// TIA Portal V17 export
// export: Created 2025-06-25T13:13:07.6103619Z, ExportSetting WithDefaults, DisplayName Totally Integrated Automation Portal, DisplayVersion V17 Update 8, DisplayName TIA Portal Openness, DisplayVersion V17 Update 8, DisplayName TIA Portal Version Control Interface, DisplayVersion V17, DisplayName STEP 7 Professional, DisplayVersion V17 Update 8, DisplayName STEP 7 Safety, DisplayVersion V17 Update 6, DisplayName WinCC Advanced, DisplayVersion V17 Update 8
FUNCTION_BLOCK "SuperheatControl"   // FB23, FBD
TITLE = Pinch setpoint from superheat
{ S7_Optimized_Access := 'TRUE' }
VERSION : 0.1
// stored: AutoNumber true, IsIECCheckEnabled false, IsRetainMemResEnabled false, MemoryReserve 100, SetENOAutomatically false, UDAEnableTagReadback false
   VAR_INPUT
      bEnable { ExternalAccessible := 'False'; ExternalVisible := 'False'; ExternalWritable := 'False'} : Bool;   // 1 = enable controller 0 = disable controller
      bReset { ExternalAccessible := 'False'; ExternalVisible := 'False'; ExternalWritable := 'False'} : Bool;   // 1 = reset manual mode
      AdditionalSuperheat { ExternalAccessible := 'False'; ExternalVisible := 'False'; ExternalWritable := 'False'} : Real;
   END_VAR
   VAR_OUTPUT
      AddSuperheat { ExternalAccessible := 'False'; ExternalVisible := 'False'; ExternalWritable := 'False'} : Real;
   END_VAR
   VAR
      SuperheatSetpoint { ExternalAccessible := 'False'; ExternalVisible := 'False'; ExternalWritable := 'False'} : Real;
      PinchSetpoint { ExternalAccessible := 'False'; ExternalVisible := 'False'; ExternalWritable := 'False'} : Real;
      PinchPerformanceCurrent { ExternalAccessible := 'False'; ExternalVisible := 'False'; ExternalWritable := 'False'} : Real;
      Regulator { ExternalAccessible := 'False'; ExternalVisible := 'False'; ExternalWritable := 'False'} : Struct
         x_intern_1 { ExternalAccessible := 'False'; ExternalVisible := 'False'; ExternalWritable := 'False'} : Real;
         x_intern_2 { ExternalAccessible := 'False'; ExternalVisible := 'False'; ExternalWritable := 'False'} : Real;
         x_intern_3 { ExternalAccessible := 'False'; ExternalVisible := 'False'; ExternalWritable := 'False'} : Real;
      END_STRUCT;
      Enabled { ExternalAccessible := 'False'; ExternalVisible := 'False'; ExternalWritable := 'False'} : Bool;
      A3020 { ExternalAccessible := 'False'; ExternalVisible := 'False'; ExternalWritable := 'False'} : "fbHMIEvent";
   END_VAR
   VAR_TEMP
      PinchPerformance : Real;
      PIDControlInactive : Bool;   // Is true if pinch setpoint is externally controlled
   END_VAR
BEGIN

REGION Network 1: Reset manual mode
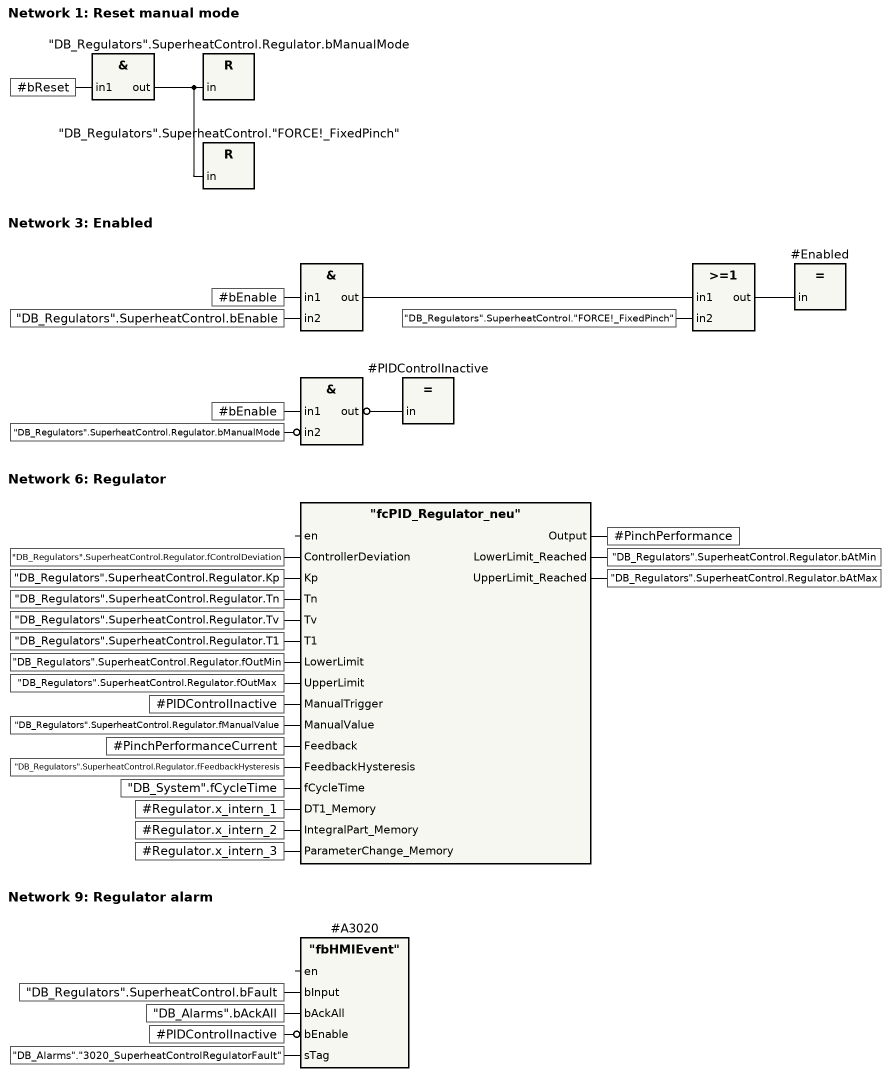
   IF #bReset THEN
       "DB_Regulators".SuperheatControl.Regulator.bManualMode := FALSE;
       "DB_Regulators".SuperheatControl."FORCE!_FixedPinch" := FALSE;
   END_IF;
END_REGION

REGION Network 2 (SCL): Manual values are given as Pinch, regulator works on "Pinch Performance"
   "DB_Regulators".SuperheatControl.Regulator.bManualMode := "DB_Regulators".SuperheatControl."FORCE!_FixedPinch";
END_REGION

REGION Network 3: Enabled
   // NOTE that we are not using the conventional bManual bit!!
   // Due to the difference between "Pinch Performance" and "Pinch"
   #Enabled := (#bEnable AND "DB_Regulators".SuperheatControl.bEnable) OR "DB_Regulators".SuperheatControl."FORCE!_FixedPinch";
   #PIDControlInactive := NOT (#bEnable AND NOT "DB_Regulators".SuperheatControl.Regulator.bManualMode);
END_REGION

REGION Network 4 (SCL): Superheat setpoint
   //Additional Superheat
   #AddSuperheat := #AdditionalSuperheat + "DB_Regulators".SuperheatControl.AdditionalSuperheat + "DB_CurrentSetting".Fluid.T_AdditionalSuperHeatEvaporator;

   #SuperheatSetpoint := 1.0 * "RecTarget"("DB_Regulators".SuperheatControl.fineTuningRecTarget) +
                         1.0 * #AddSuperheat;

   // Superheat setpoint
   IF "DB_State".State."6_Running" THEN
       #SuperheatSetpoint := #SuperheatSetpoint + 1.0 * "VapPerformance"(AddSuperheat := #AddSuperheat, Pinch := #PinchSetpoint);
   ELSE
       #SuperheatSetpoint := #SuperheatSetpoint + 0.5 * "VapPerformance"(AddSuperheat := #AddSuperheat, Pinch := #PinchSetpoint);

   END_IF;

   // Enforce a lower bound on the superheat
   #SuperheatSetpoint := MAX(IN1 := #SuperheatSetpoint, IN2 := "DB_CurrentSetting".System.Limits.T_SuperHeatCompressorIn_Min + 5.5);
END_REGION

REGION Network 5 (SCL): Deviation
   IF "DB_Regulators".SuperheatControl.Regulator.bManualMode = TRUE THEN
       "DB_Regulators".SuperheatControl.Regulator.fManualValue := LN(MAX(IN1 := "DB_Regulators".SuperheatControl."FORCE!_FixedPinch_Value", IN2 := 0.01)) * "DB_Regulators".SuperheatControl.ExponentialPinchFactor;
       "DB_Regulators".SuperheatControl.bFault := FALSE;
   ELSE
       //- Preset manual value to current pinch value to set controller to this value if inactive. Except if bManualMode whwre we directely set it to the target pinch performance
       //- Limited to 1K superhetat to prevent division by zero and critical low pinch values
       "DB_Regulators".SuperheatControl.Regulator.fManualValue := LN(MAX(IN1 := "DB_Calc".HeatSource.Pinch.fValue, IN2 := 1)) * "DB_Regulators".SuperheatControl.ExponentialPinchFactor;

       //Preset with current pinch as starting value if "FORCE!_FixedPinch is used
       "DB_Regulators".SuperheatControl."FORCE!_FixedPinch_Value" := "DB_Calc".HeatSource.Pinch.fValue;


       //Auto mode setpoint
       IF "isNaN"("DB_Calc".LowPressPart.CompressorSuperheat.fValue) OR "isNaN"(#SuperheatSetpoint) THEN
           "DB_Regulators".SuperheatControl.Regulator.fControlDeviation := 0;
           "DB_Regulators".SuperheatControl.bFault := TRUE;
       ELSE
           "DB_Regulators".SuperheatControl.Regulator.fControlDeviation := #SuperheatSetpoint - "DB_Calc".LowPressPart.CompressorSuperheat.fValue;
           "DB_Regulators".SuperheatControl.bFault := FALSE;
       END_IF;
   END_IF;

   //- Current pinch performance for informative reasons
   //- Limited to 0.1K to prevent division by zero 
   #PinchPerformanceCurrent := LN(MAX(IN1 := "DB_Calc".HeatSource.Pinch.fValue, IN2 := 0.1)) * "DB_Regulators".SuperheatControl.ExponentialPinchFactor;
END_REGION

REGION Network 6: Regulator
   "fcPID_Regulator_neu"(ControllerDeviation := "DB_Regulators".SuperheatControl.Regulator.fControlDeviation,
                         Kp := "DB_Regulators".SuperheatControl.Regulator.Kp,
                         Tn := "DB_Regulators".SuperheatControl.Regulator.Tn,
                         Tv := "DB_Regulators".SuperheatControl.Regulator.Tv,
                         T1 := "DB_Regulators".SuperheatControl.Regulator.T1,
                         LowerLimit := "DB_Regulators".SuperheatControl.Regulator.fOutMin,
                         UpperLimit := "DB_Regulators".SuperheatControl.Regulator.fOutMax,
                         ManualTrigger := #PIDControlInactive,
                         ManualValue := "DB_Regulators".SuperheatControl.Regulator.fManualValue,
                         Feedback := #PinchPerformanceCurrent,
                         FeedbackHysteresis := "DB_Regulators".SuperheatControl.Regulator.fFeedbackHysteresis,
                         fCycleTime := "DB_System".fCycleTime,
                         DT1_Memory := #Regulator.x_intern_1,
                         IntegralPart_Memory := #Regulator.x_intern_2,
                         ParameterChange_Memory := #Regulator.x_intern_3,
                         Output => #PinchPerformance,
                         LowerLimit_Reached => "DB_Regulators".SuperheatControl.Regulator.bAtMin,
                         UpperLimit_Reached => "DB_Regulators".SuperheatControl.Regulator.bAtMax);
END_REGION

REGION Network 7 (SCL): Convert Pinch Performance to Pinch
   //The PinchPerfomance value is interpreted logarithmically as pinch set point (-oo => 0K; 0 => 1K; 110 => 163K). 
   //Constant changes of PinchPerformance will cause only relative changes of the effective pinch. Pinch = e^(PinchPerformance/21,6)
   IF "DB_Regulators".SuperheatControl.Regulator.bManualMode = TRUE THEN
       "DB_Regulators".SuperheatControl.Regulator.fOut := "DB_Regulators".SuperheatControl."FORCE!_FixedPinch_Value";
   ELSE
       "DB_Regulators".SuperheatControl.Regulator.fOut := EXP(#PinchPerformance / "DB_Regulators".SuperheatControl.ExponentialPinchFactor);
       // Keep the manual value in sync to avoid discontinuities when switching from normal operation to Manual:
       //"DB_Regulators".SuperheatControl."FORCE!_FixedPinch_Value" := "DB_Regulators".SuperheatControl.Regulator.fOut;

   END_IF;
END_REGION

REGION Network 8 (SCL): Disable
   //IF #Enabled = FALSE THEN
   //    "DB_Regulators".SuperheatControl.Regulator.fOut := "DB_Regulators".SuperheatControl."FORCE!_FixedPinch_Value";
   //    "DB_Regulators".SuperheatControl.Regulator.bAtMin := FALSE;
   //    "DB_Regulators".SuperheatControl.Regulator.bAtMax := FALSE;
   //END_IF;
END_REGION

REGION Network 9: Regulator alarm
   #A3020(bInput := "DB_Regulators".SuperheatControl.bFault,   // "fbHMIEvent"
          bAckAll := "DB_Alarms".bAckAll,
          bEnable := NOT #PIDControlInactive,
          sTag := "DB_Alarms"."3020_SuperheatControlRegulatorFault");
END_REGION

REGION Network 10 (SCL): Mode
   // Only Auto or Manual in this regulator
   // Mode
   IF "DB_Regulators".SuperheatControl."FORCE!_FixedPinch" = TRUE THEN
       "DB_Regulators".SuperheatControl.nMode := 2;
   ELSE
       "DB_Regulators".SuperheatControl.nMode := 1;
   END_IF;
END_REGION
END_FUNCTION_BLOCK
